Staubli VAL3: set.pgx

public program set(string x_sItem, num x_nIndex)
begin
  // set the name
  // saveAxis[x_nIndex].sName=x_sItem
  sSaveaxis[x_nIndex]=x_sItem
end
